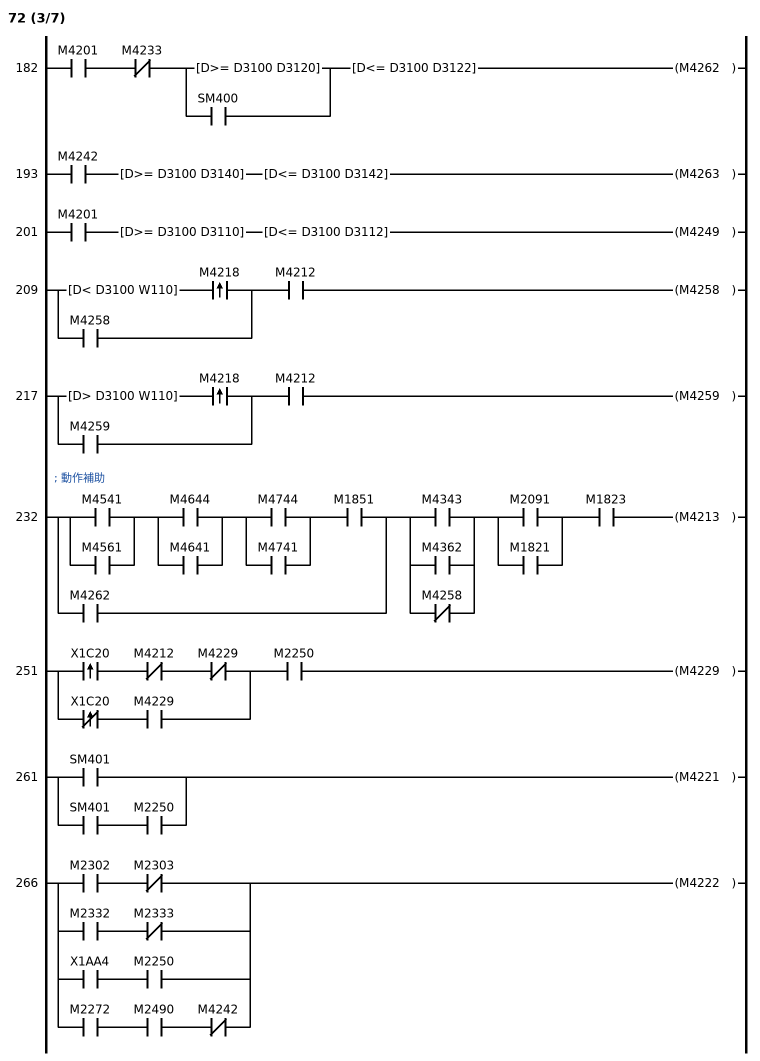
182   LD      M4201
      ANI     M4233
      LDD>=   D3100 D3120
      OR      SM400
      ANB
      ANDD<=  D3100 D3122
      OUT     M4262
193   LD      M4242
      ANDD>=  D3100 D3140
      ANDD<=  D3100 D3142
      OUT     M4263
201   LD      M4201
      ANDD>=  D3100 D3110
      ANDD<=  D3100 D3112
      OUT     M4249
209   LDD<    D3100 W110
      ANDP    M4218
      OR      M4258
      AND     M4212
      OUT     M4258
217   LDD>    D3100 W110
      ANDP    M4218
      OR      M4259
      AND     M4212
      OUT     M4259
; 動作補助
232   LD      M4541
      OR      M4561
      LD      M4644
      OR      M4641
      ANB
      LD      M4744
      OR      M4741
      ANB
      AND     M1851
      OR      M4262
      LD      M4343
      OR      M4362
      ORI     M4258
      ANB
      LD      M2091
      OR      M1821
      ANB
      AND     M1823
      OUT     M4213
251   LDP     X1C20
      ANI     M4212
      ANI     M4229
      LDPI    X1C20
      AND     M4229
      ORB
      AND     M2250
      OUT     M4229
261   LD      SM401
      LD      SM401
      AND     M2250
      ORB
      OUT     M4221
266   LD      M2302
      ANI     M2303
      LD      M2332
      ANI     M2333
      ORB
      LD      X1AA4
      AND     M2250
      ORB
      LD      M2272
      AND     M2490
      ANI     M4242
      ORB
      OUT     M4222
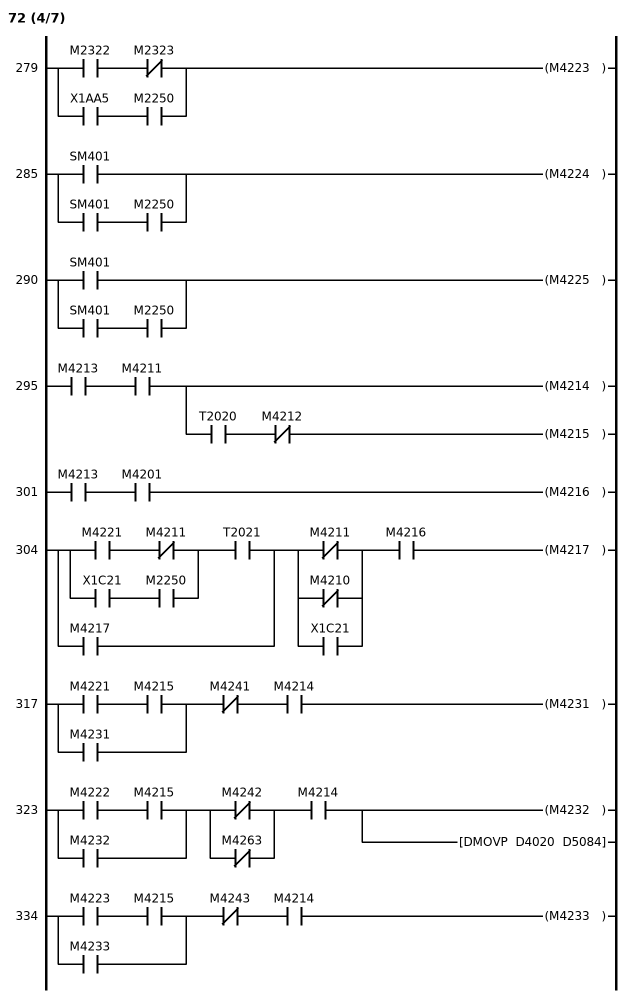
279   LD      M2322
      ANI     M2323
      LD      X1AA5
      AND     M2250
      ORB
      OUT     M4223
285   LD      SM401
      LD      SM401
      AND     M2250
      ORB
      OUT     M4224
290   LD      SM401
      LD      SM401
      AND     M2250
      ORB
      OUT     M4225
295   LD      M4213
      AND     M4211
      OUT     M4214
      AND     T2020
      ANI     M4212
      OUT     M4215
301   LD      M4213
      AND     M4201
      OUT     M4216
304   LD      M4221
      ANI     M4211
      LD      X1C21
      AND     M2250
      ORB
      AND     T2021
      OR      M4217
      LDI     M4211
      ORI     M4210
      OR      X1C21
      ANB
      AND     M4216
      OUT     M4217
317   LD      M4221
      AND     M4215
      OR      M4231
      ANI     M4241
      AND     M4214
      OUT     M4231
323   LD      M4222
      AND     M4215
      OR      M4232
      LDI     M4242
      ORI     M4263
      ANB
      AND     M4214
      OUT     M4232
      DMOVP   D4020 D5084
334   LD      M4223
      AND     M4215
      OR      M4233
      ANI     M4243
      AND     M4214
      OUT     M4233
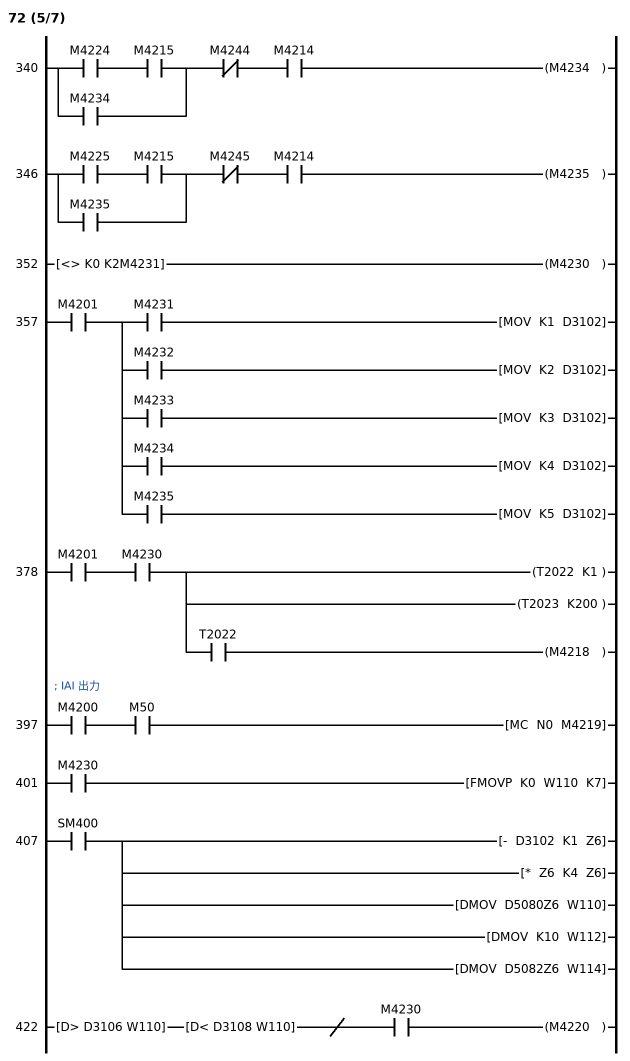
340   LD      M4224
      AND     M4215
      OR      M4234
      ANI     M4244
      AND     M4214
      OUT     M4234
346   LD      M4225
      AND     M4215
      OR      M4235
      ANI     M4245
      AND     M4214
      OUT     M4235
352   LD<>    K0 K2M4231
      OUT     M4230
357   LD      M4201
      MPS
      AND     M4231
      MOV     K1 D3102
      MRD
      AND     M4232
      MOV     K2 D3102
      MRD
      AND     M4233
      MOV     K3 D3102
      MRD
      AND     M4234
      MOV     K4 D3102
      MPP
      AND     M4235
      MOV     K5 D3102
378   LD      M4201
      AND     M4230
      OUT     T2022 K1
      OUT     T2023 K200
      AND     T2022
      OUT     M4218
; IAI 出力
397   LD      M4200
      AND     M50
      MC      N0 M4219
401   LD      M4230
      FMOVP   K0 W110 K7
407   LD      SM400
      -       D3102 K1 Z6
      *       Z6 K4 Z6
      DMOV    D5080Z6 W110
      DMOV    K10 W112
      DMOV    D5082Z6 W114
422   LDD>    D3106 W110
      ANDD<   D3108 W110
      INV
      AND     M4230
      OUT     M4220
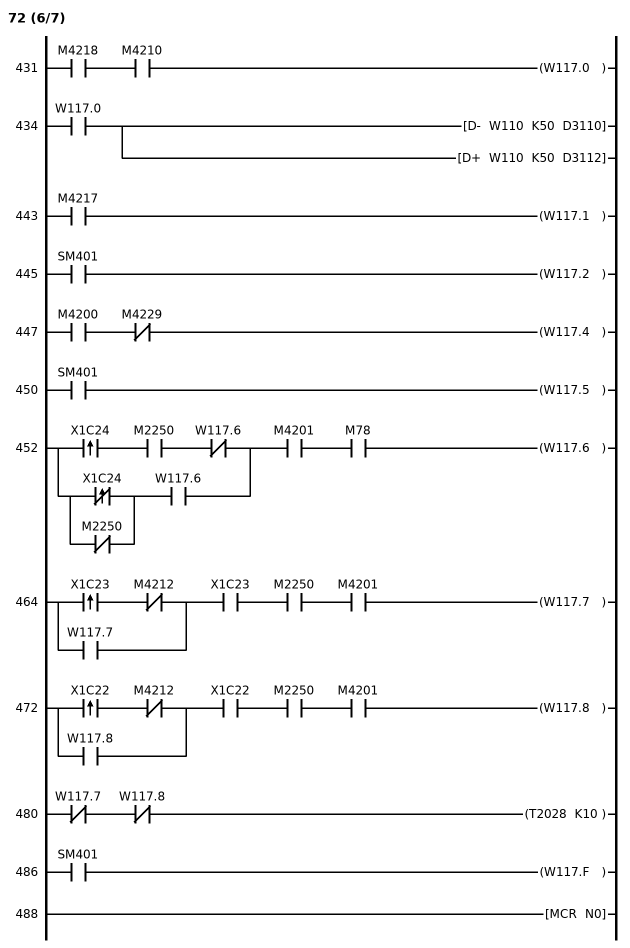
431   LD      M4218
      AND     M4210
      OUT     W117.0
434   LD      W117.0
      D-      W110 K50 D3110
      D+      W110 K50 D3112
443   LD      M4217
      OUT     W117.1
445   LD      SM401
      OUT     W117.2
447   LD      M4200
      ANI     M4229
      OUT     W117.4
450   LD      SM401
      OUT     W117.5
452   LDP     X1C24
      AND     M2250
      ANI     W117.6
      LDPI    X1C24
      ORI     M2250
      AND     W117.6
      ORB
      AND     M4201
      AND     M78
      OUT     W117.6
464   LDP     X1C23
      ANI     M4212
      OR      W117.7
      AND     X1C23
      AND     M2250
      AND     M4201
      OUT     W117.7
472   LDP     X1C22
      ANI     M4212
      OR      W117.8
      AND     X1C22
      AND     M2250
      AND     M4201
      OUT     W117.8
480   LDI     W117.7
      ANI     W117.8
      OUT     T2028 K10
486   LD      SM401
      OUT     W117.F
488   MCR     N0
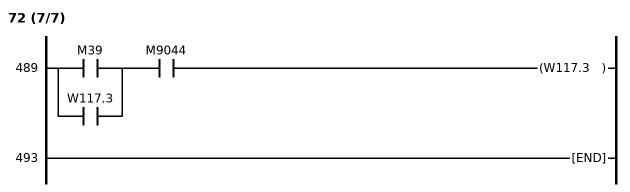
489   LD      M39
      OR      W117.3
      AND     M9044
      OUT     W117.3
493   END
END_PROGRAM

PROGRAM 73
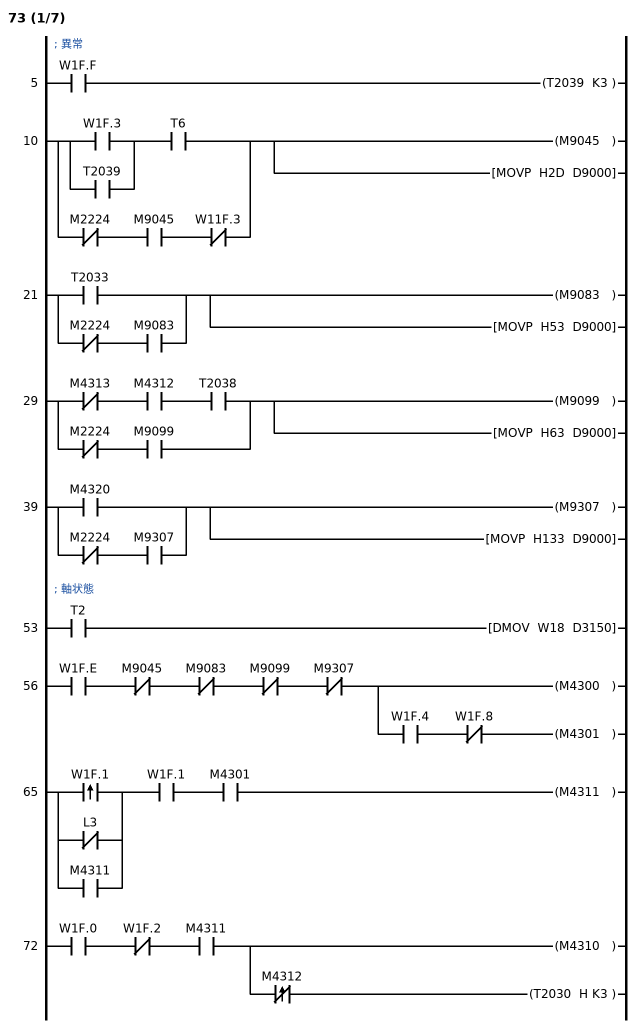
; 異常
5     LD      W1F.F
      OUT     T2039 K3
10    LD      W1F.3
      OR      T2039
      AND     T6
      LDI     M2224
      AND     M9045
      ANI     W11F.3
      ORB
      OUT     M9045
      MOVP    H2D D9000
21    LD      T2033
      LDI     M2224
      AND     M9083
      ORB
      OUT     M9083
      MOVP    H53 D9000
29    LDI     M4313
      AND     M4312
      AND     T2038
      LDI     M2224
      AND     M9099
      ORB
      OUT     M9099
      MOVP    H63 D9000
39    LD      M4320
      LDI     M2224
      AND     M9307
      ORB
      OUT     M9307
      MOVP    H133 D9000
; 軸状態
53    LD      T2
      DMOV    W18 D3150
56    LD      W1F.E
      ANI     M9045
      ANI     M9083
      ANI     M9099
      ANI     M9307
      OUT     M4300
      AND     W1F.4
      ANI     W1F.8
      OUT     M4301
65    LDP     W1F.1
      ORI     L3
      OR      M4311
      AND     W1F.1
      AND     M4301
      OUT     M4311
72    LD      W1F.0
      ANI     W1F.2
      AND     M4311
      OUT     M4310
      ANDPI   M4312
      OUTH    T2030 K3
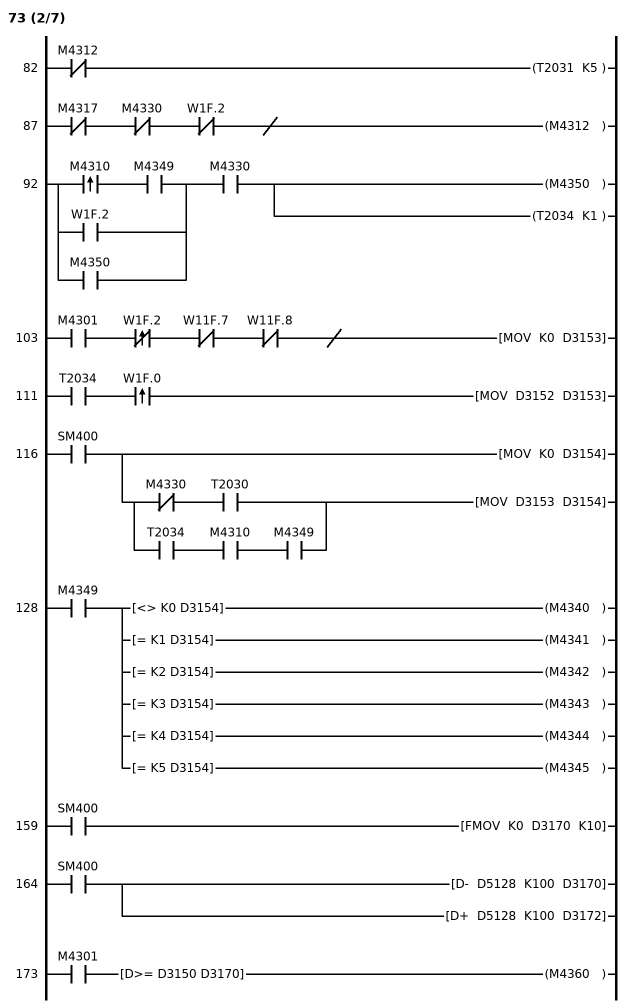
82    LDI     M4312
      OUT     T2031 K5
87    LDI     M4317
      ANI     M4330
      ANI     W1F.2
      INV
      OUT     M4312
92    LDP     M4310
      AND     M4349
      OR      W1F.2
      OR      M4350
      AND     M4330
      OUT     M4350
      OUT     T2034 K1
103   LD      M4301
      ANDPI   W1F.2
      ANI     W11F.7
      ANI     W11F.8
      INV
      MOV     K0 D3153
111   LD      T2034
      ANDP    W1F.0
      MOV     D3152 D3153
116   LD      SM400
      MOV     K0 D3154
      LDI     M4330
      AND     T2030
      LD      T2034
      AND     M4310
      AND     M4349
      ORB
      ANB
      MOV     D3153 D3154
128   LD      M4349
      MPS
      AND<>   K0 D3154
      OUT     M4340
      MRD
      AND=    K1 D3154
      OUT     M4341
      MRD
      AND=    K2 D3154
      OUT     M4342
      MRD
      AND=    K3 D3154
      OUT     M4343
      MRD
      AND=    K4 D3154
      OUT     M4344
      MPP
      AND=    K5 D3154
      OUT     M4345
159   LD      SM400
      FMOV    K0 D3170 K10
164   LD      SM400
      D-      D5128 K100 D3170
      D+      D5128 K100 D3172
173   LD      M4301
      ANDD>=  D3150 D3170
      OUT     M4360
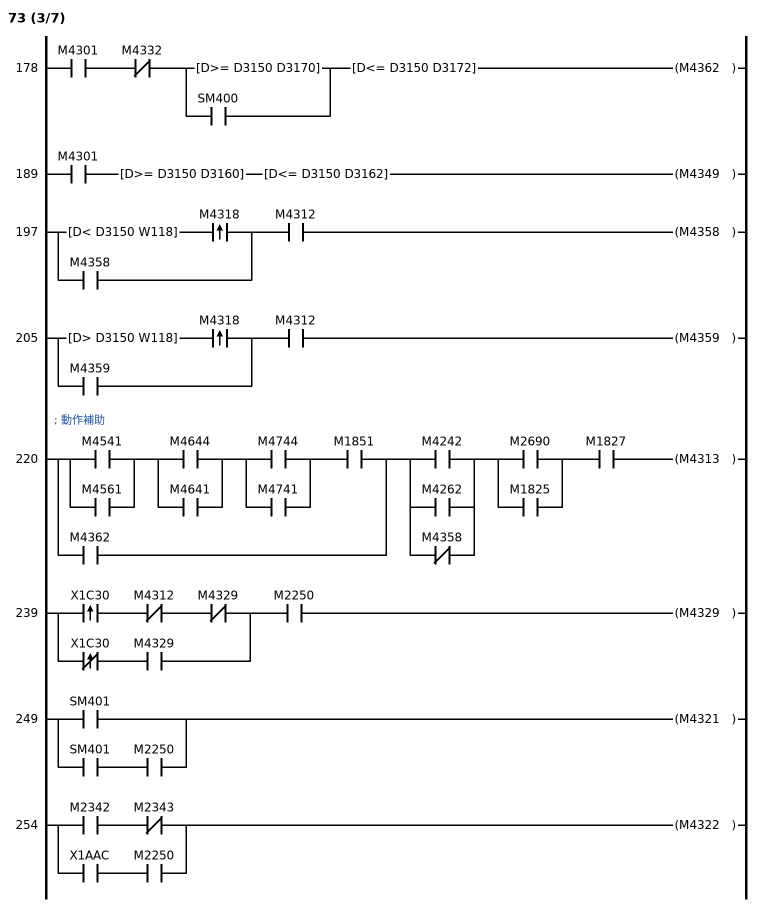
178   LD      M4301
      ANI     M4332
      LDD>=   D3150 D3170
      OR      SM400
      ANB
      ANDD<=  D3150 D3172
      OUT     M4362
189   LD      M4301
      ANDD>=  D3150 D3160
      ANDD<=  D3150 D3162
      OUT     M4349
197   LDD<    D3150 W118
      ANDP    M4318
      OR      M4358
      AND     M4312
      OUT     M4358
205   LDD>    D3150 W118
      ANDP    M4318
      OR      M4359
      AND     M4312
      OUT     M4359
; 動作補助
220   LD      M4541
      OR      M4561
      LD      M4644
      OR      M4641
      ANB
      LD      M4744
      OR      M4741
      ANB
      AND     M1851
      OR      M4362
      LD      M4242
      OR      M4262
      ORI     M4358
      ANB
      LD      M2690
      OR      M1825
      ANB
      AND     M1827
      OUT     M4313
239   LDP     X1C30
      ANI     M4312
      ANI     M4329
      LDPI    X1C30
      AND     M4329
      ORB
      AND     M2250
      OUT     M4329
249   LD      SM401
      LD      SM401
      AND     M2250
      ORB
      OUT     M4321
254   LD      M2342
      ANI     M2343
      LD      X1AAC
      AND     M2250
      ORB
      OUT     M4322
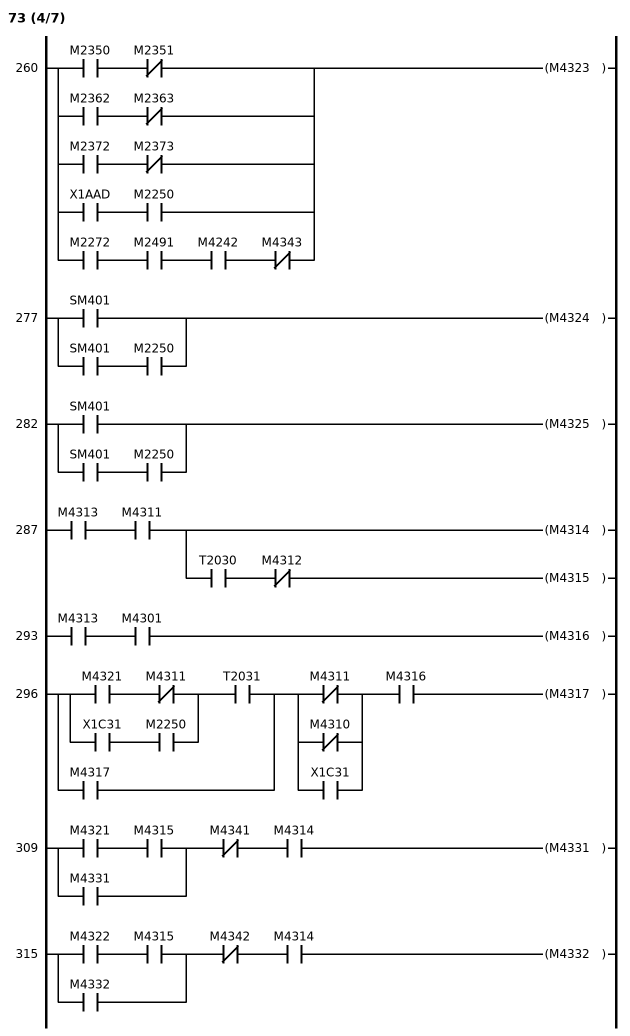
260   LD      M2350
      ANI     M2351
      LD      M2362
      ANI     M2363
      ORB
      LD      M2372
      ANI     M2373
      ORB
      LD      X1AAD
      AND     M2250
      ORB
      LD      M2272
      AND     M2491
      AND     M4242
      ANI     M4343
      ORB
      OUT     M4323
277   LD      SM401
      LD      SM401
      AND     M2250
      ORB
      OUT     M4324
282   LD      SM401
      LD      SM401
      AND     M2250
      ORB
      OUT     M4325
287   LD      M4313
      AND     M4311
      OUT     M4314
      AND     T2030
      ANI     M4312
      OUT     M4315
293   LD      M4313
      AND     M4301
      OUT     M4316
296   LD      M4321
      ANI     M4311
      LD      X1C31
      AND     M2250
      ORB
      AND     T2031
      OR      M4317
      LDI     M4311
      ORI     M4310
      OR      X1C31
      ANB
      AND     M4316
      OUT     M4317
309   LD      M4321
      AND     M4315
      OR      M4331
      ANI     M4341
      AND     M4314
      OUT     M4331
315   LD      M4322
      AND     M4315
      OR      M4332
      ANI     M4342
      AND     M4314
      OUT     M4332
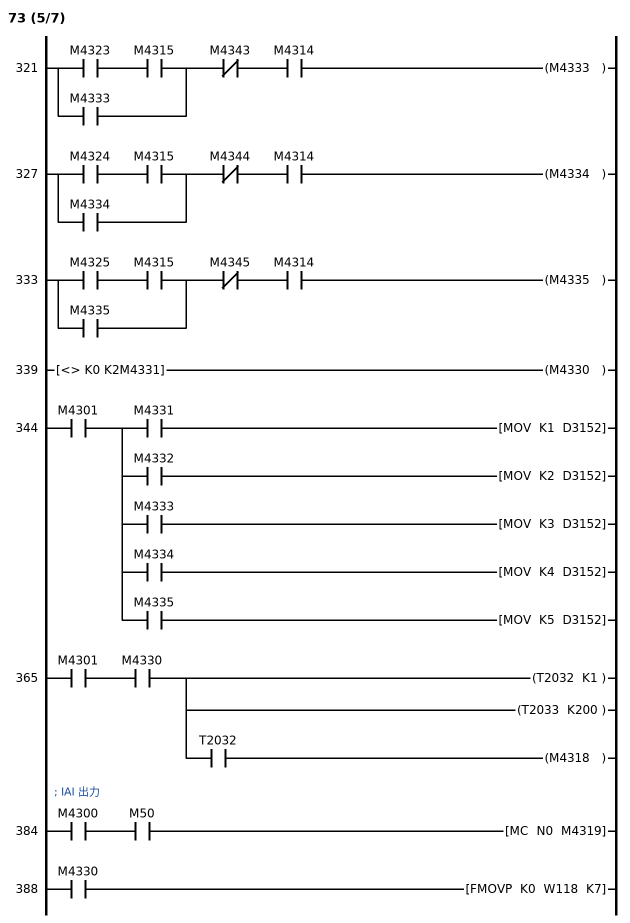
321   LD      M4323
      AND     M4315
      OR      M4333
      ANI     M4343
      AND     M4314
      OUT     M4333
327   LD      M4324
      AND     M4315
      OR      M4334
      ANI     M4344
      AND     M4314
      OUT     M4334
333   LD      M4325
      AND     M4315
      OR      M4335
      ANI     M4345
      AND     M4314
      OUT     M4335
339   LD<>    K0 K2M4331
      OUT     M4330
344   LD      M4301
      MPS
      AND     M4331
      MOV     K1 D3152
      MRD
      AND     M4332
      MOV     K2 D3152
      MRD
      AND     M4333
      MOV     K3 D3152
      MRD
      AND     M4334
      MOV     K4 D3152
      MPP
      AND     M4335
      MOV     K5 D3152
365   LD      M4301
      AND     M4330
      OUT     T2032 K1
      OUT     T2033 K200
      AND     T2032
      OUT     M4318
; IAI 出力
384   LD      M4300
      AND     M50
      MC      N0 M4319
388   LD      M4330
      FMOVP   K0 W118 K7
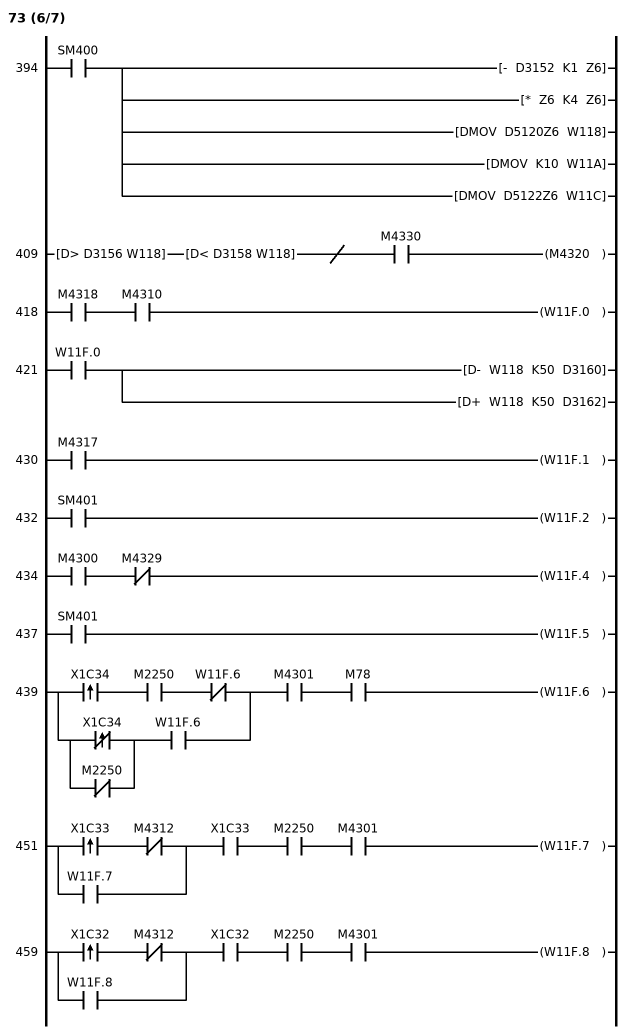
394   LD      SM400
      -       D3152 K1 Z6
      *       Z6 K4 Z6
      DMOV    D5120Z6 W118
      DMOV    K10 W11A
      DMOV    D5122Z6 W11C
409   LDD>    D3156 W118
      ANDD<   D3158 W118
      INV
      AND     M4330
      OUT     M4320
418   LD      M4318
      AND     M4310
      OUT     W11F.0
421   LD      W11F.0
      D-      W118 K50 D3160
      D+      W118 K50 D3162
430   LD      M4317
      OUT     W11F.1
432   LD      SM401
      OUT     W11F.2
434   LD      M4300
      ANI     M4329
      OUT     W11F.4
437   LD      SM401
      OUT     W11F.5
439   LDP     X1C34
      AND     M2250
      ANI     W11F.6
      LDPI    X1C34
      ORI     M2250
      AND     W11F.6
      ORB
      AND     M4301
      AND     M78
      OUT     W11F.6
451   LDP     X1C33
      ANI     M4312
      OR      W11F.7
      AND     X1C33
      AND     M2250
      AND     M4301
      OUT     W11F.7
459   LDP     X1C32
      ANI     M4312
      OR      W11F.8
      AND     X1C32
      AND     M2250
      AND     M4301
      OUT     W11F.8
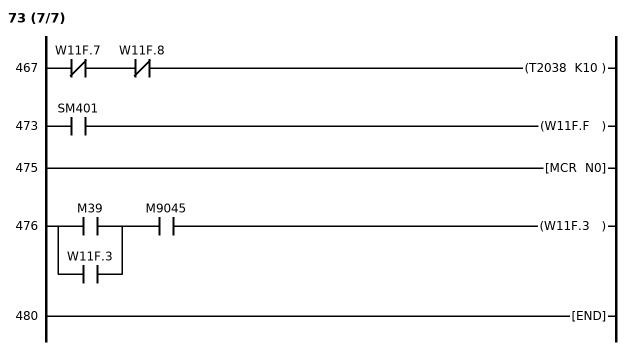
467   LDI     W11F.7
      ANI     W11F.8
      OUT     T2038 K10
473   LD      SM401
      OUT     W11F.F
475   MCR     N0
476   LD      M39
      OR      W11F.3
      AND     M9045
      OUT     W11F.3
480   END
END_PROGRAM

PROGRAM 74
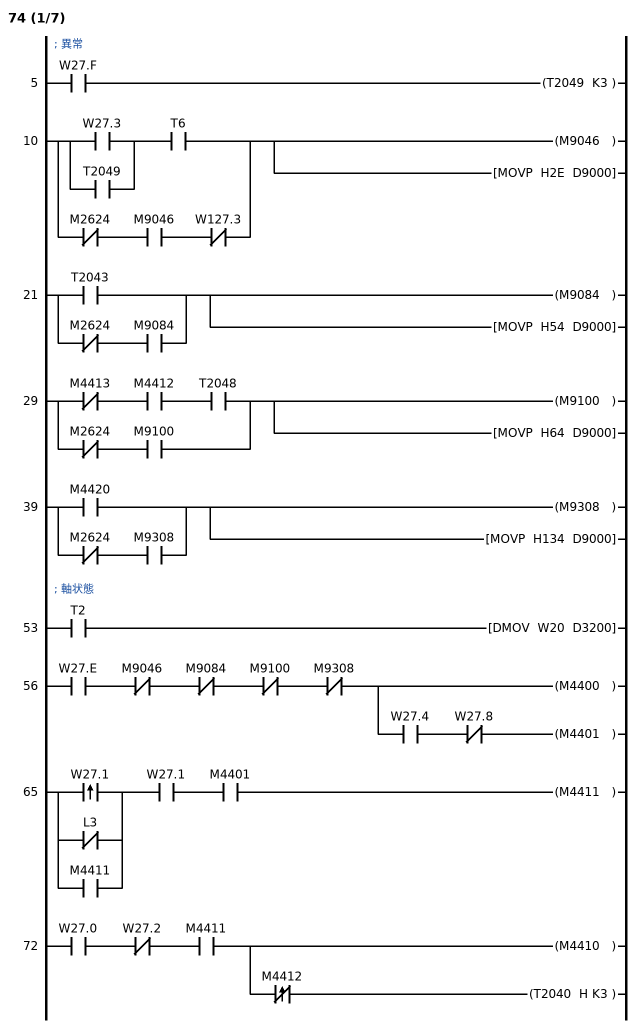
; 異常
5     LD      W27.F
      OUT     T2049 K3
10    LD      W27.3
      OR      T2049
      AND     T6
      LDI     M2624
      AND     M9046
      ANI     W127.3
      ORB
      OUT     M9046
      MOVP    H2E D9000
21    LD      T2043
      LDI     M2624
      AND     M9084
      ORB
      OUT     M9084
      MOVP    H54 D9000
29    LDI     M4413
      AND     M4412
      AND     T2048
      LDI     M2624
      AND     M9100
      ORB
      OUT     M9100
      MOVP    H64 D9000
39    LD      M4420
      LDI     M2624
      AND     M9308
      ORB
      OUT     M9308
      MOVP    H134 D9000
; 軸状態
53    LD      T2
      DMOV    W20 D3200
56    LD      W27.E
      ANI     M9046
      ANI     M9084
      ANI     M9100
      ANI     M9308
      OUT     M4400
      AND     W27.4
      ANI     W27.8
      OUT     M4401
65    LDP     W27.1
      ORI     L3
      OR      M4411
      AND     W27.1
      AND     M4401
      OUT     M4411
72    LD      W27.0
      ANI     W27.2
      AND     M4411
      OUT     M4410
      ANDPI   M4412
      OUTH    T2040 K3
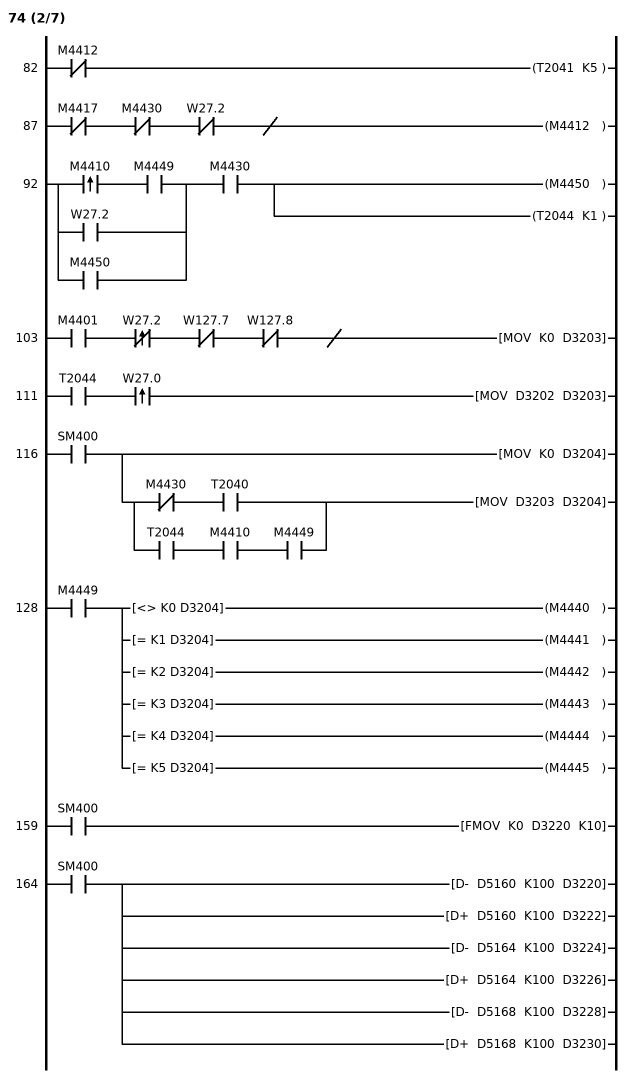
82    LDI     M4412
      OUT     T2041 K5
87    LDI     M4417
      ANI     M4430
      ANI     W27.2
      INV
      OUT     M4412
92    LDP     M4410
      AND     M4449
      OR      W27.2
      OR      M4450
      AND     M4430
      OUT     M4450
      OUT     T2044 K1
103   LD      M4401
      ANDPI   W27.2
      ANI     W127.7
      ANI     W127.8
      INV
      MOV     K0 D3203
111   LD      T2044
      ANDP    W27.0
      MOV     D3202 D3203
116   LD      SM400
      MOV     K0 D3204
      LDI     M4430
      AND     T2040
      LD      T2044
      AND     M4410
      AND     M4449
      ORB
      ANB
      MOV     D3203 D3204
128   LD      M4449
      MPS
      AND<>   K0 D3204
      OUT     M4440
      MRD
      AND=    K1 D3204
      OUT     M4441
      MRD
      AND=    K2 D3204
      OUT     M4442
      MRD
      AND=    K3 D3204
      OUT     M4443
      MRD
      AND=    K4 D3204
      OUT     M4444
      MPP
      AND=    K5 D3204
      OUT     M4445
159   LD      SM400
      FMOV    K0 D3220 K10
164   LD      SM400
      D-      D5160 K100 D3220
      D+      D5160 K100 D3222
      D-      D5164 K100 D3224
      D+      D5164 K100 D3226
      D-      D5168 K100 D3228
      D+      D5168 K100 D3230
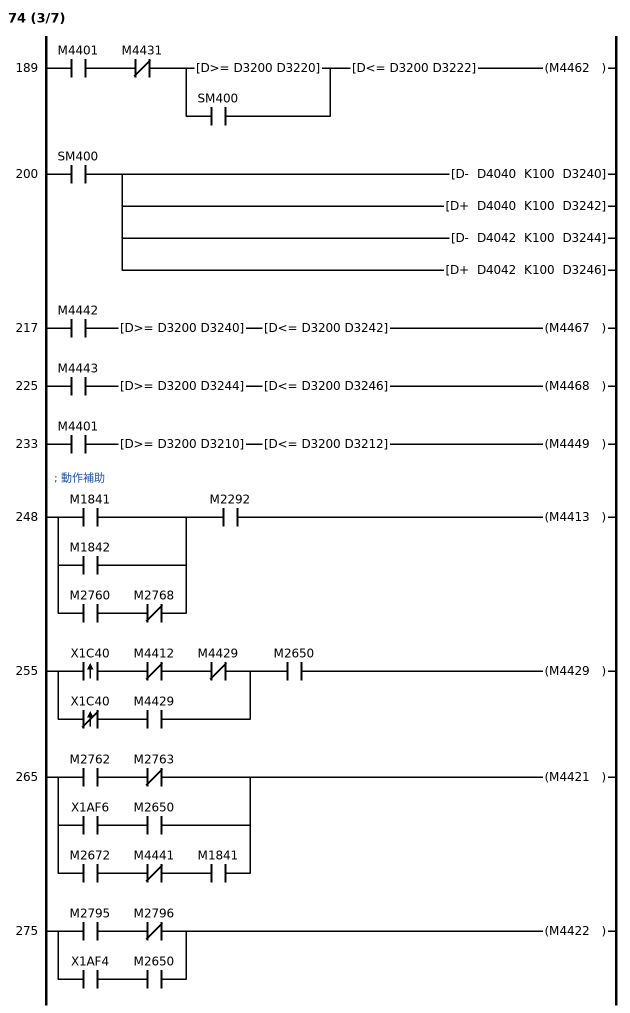
189   LD      M4401
      ANI     M4431
      LDD>=   D3200 D3220
      OR      SM400
      ANB
      ANDD<=  D3200 D3222
      OUT     M4462
200   LD      SM400
      D-      D4040 K100 D3240
      D+      D4040 K100 D3242
      D-      D4042 K100 D3244
      D+      D4042 K100 D3246
217   LD      M4442
      ANDD>=  D3200 D3240
      ANDD<=  D3200 D3242
      OUT     M4467
225   LD      M4443
      ANDD>=  D3200 D3244
      ANDD<=  D3200 D3246
      OUT     M4468
233   LD      M4401
      ANDD>=  D3200 D3210
      ANDD<=  D3200 D3212
      OUT     M4449
; 動作補助
248   LD      M1841
      OR      M1842
      LD      M2760
      ANI     M2768
      ORB
      AND     M2292
      OUT     M4413
255   LDP     X1C40
      ANI     M4412
      ANI     M4429
      LDPI    X1C40
      AND     M4429
      ORB
      AND     M2650
      OUT     M4429
265   LD      M2762
      ANI     M2763
      LD      X1AF6
      AND     M2650
      ORB
      LD      M2672
      ANI     M4441
      AND     M1841
      ORB
      OUT     M4421
275   LD      M2795
      ANI     M2796
      LD      X1AF4
      AND     M2650
      ORB
      OUT     M4422
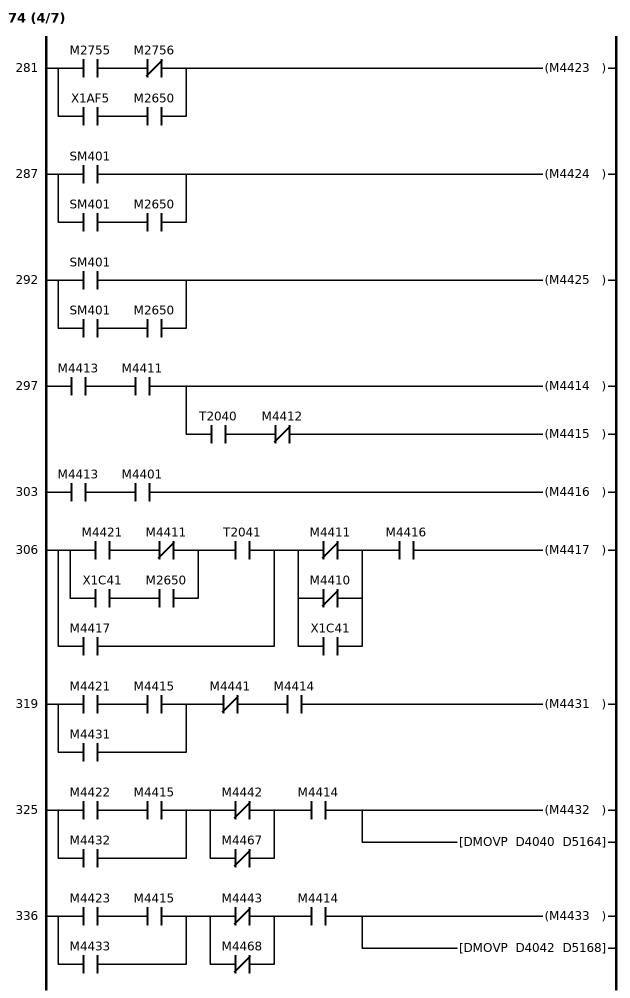
281   LD      M2755
      ANI     M2756
      LD      X1AF5
      AND     M2650
      ORB
      OUT     M4423
287   LD      SM401
      LD      SM401
      AND     M2650
      ORB
      OUT     M4424
292   LD      SM401
      LD      SM401
      AND     M2650
      ORB
      OUT     M4425
297   LD      M4413
      AND     M4411
      OUT     M4414
      AND     T2040
      ANI     M4412
      OUT     M4415
303   LD      M4413
      AND     M4401
      OUT     M4416
306   LD      M4421
      ANI     M4411
      LD      X1C41
      AND     M2650
      ORB
      AND     T2041
      OR      M4417
      LDI     M4411
      ORI     M4410
      OR      X1C41
      ANB
      AND     M4416
      OUT     M4417
319   LD      M4421
      AND     M4415
      OR      M4431
      ANI     M4441
      AND     M4414
      OUT     M4431
325   LD      M4422
      AND     M4415
      OR      M4432
      LDI     M4442
      ORI     M4467
      ANB
      AND     M4414
      OUT     M4432
      DMOVP   D4040 D5164
336   LD      M4423
      AND     M4415
      OR      M4433
      LDI     M4443
      ORI     M4468
      ANB
      AND     M4414
      OUT     M4433
      DMOVP   D4042 D5168
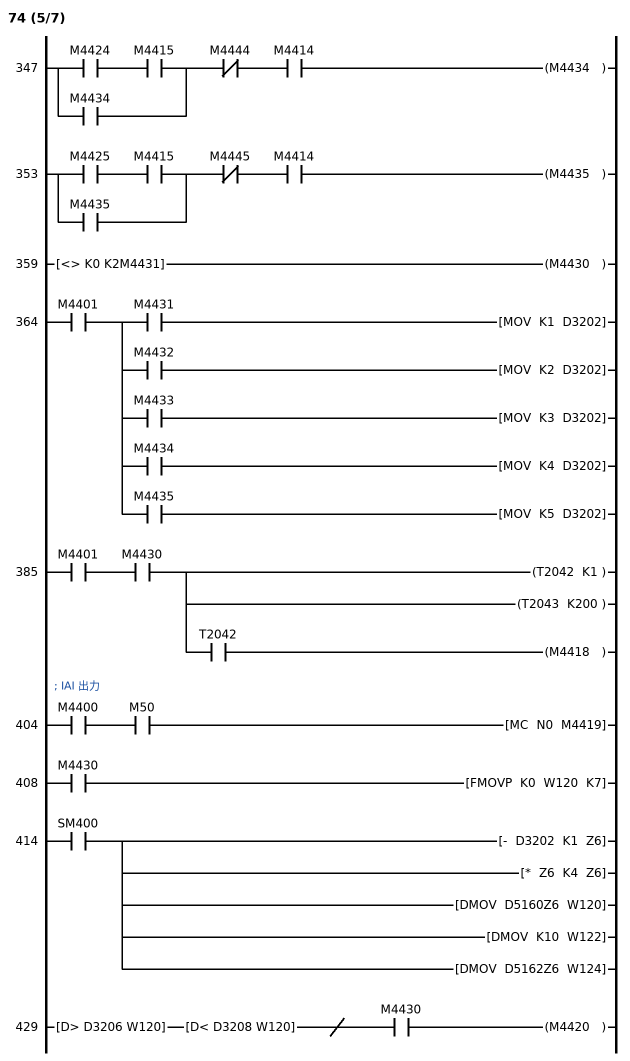
347   LD      M4424
      AND     M4415
      OR      M4434
      ANI     M4444
      AND     M4414
      OUT     M4434
353   LD      M4425
      AND     M4415
      OR      M4435
      ANI     M4445
      AND     M4414
      OUT     M4435
359   LD<>    K0 K2M4431
      OUT     M4430
364   LD      M4401
      MPS
      AND     M4431
      MOV     K1 D3202
      MRD
      AND     M4432
      MOV     K2 D3202
      MRD
      AND     M4433
      MOV     K3 D3202
      MRD
      AND     M4434
      MOV     K4 D3202
      MPP
      AND     M4435
      MOV     K5 D3202
385   LD      M4401
      AND     M4430
      OUT     T2042 K1
      OUT     T2043 K200
      AND     T2042
      OUT     M4418
; IAI 出力
404   LD      M4400
      AND     M50
      MC      N0 M4419
408   LD      M4430
      FMOVP   K0 W120 K7
414   LD      SM400
      -       D3202 K1 Z6
      *       Z6 K4 Z6
      DMOV    D5160Z6 W120
      DMOV    K10 W122
      DMOV    D5162Z6 W124
429   LDD>    D3206 W120
      ANDD<   D3208 W120
      INV
      AND     M4430
      OUT     M4420
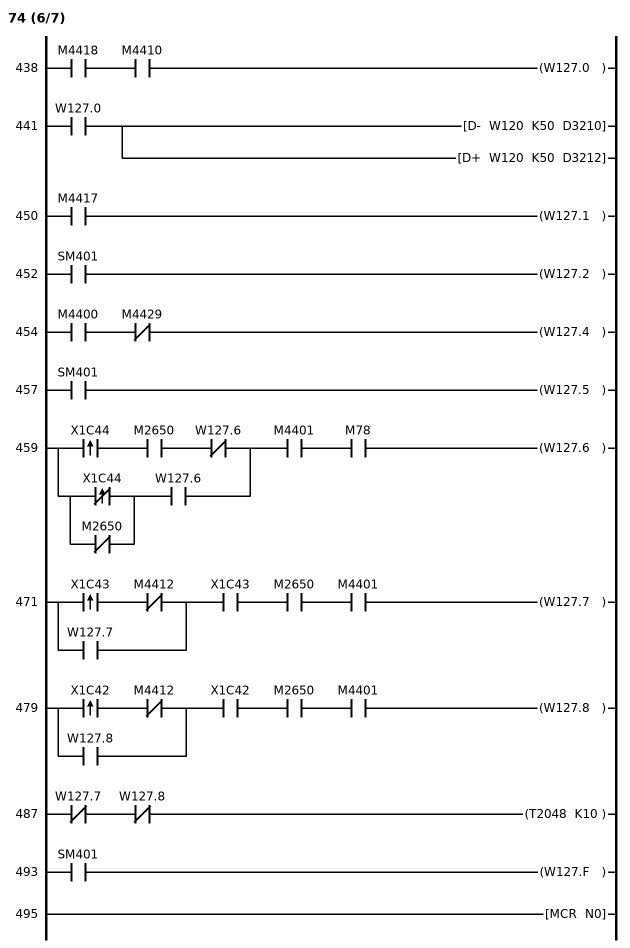
438   LD      M4418
      AND     M4410
      OUT     W127.0
441   LD      W127.0
      D-      W120 K50 D3210
      D+      W120 K50 D3212
450   LD      M4417
      OUT     W127.1
452   LD      SM401
      OUT     W127.2
454   LD      M4400
      ANI     M4429
      OUT     W127.4
457   LD      SM401
      OUT     W127.5
459   LDP     X1C44
      AND     M2650
      ANI     W127.6
      LDPI    X1C44
      ORI     M2650
      AND     W127.6
      ORB
      AND     M4401
      AND     M78
      OUT     W127.6
471   LDP     X1C43
      ANI     M4412
      OR      W127.7
      AND     X1C43
      AND     M2650
      AND     M4401
      OUT     W127.7
479   LDP     X1C42
      ANI     M4412
      OR      W127.8
      AND     X1C42
      AND     M2650
      AND     M4401
      OUT     W127.8
487   LDI     W127.7
      ANI     W127.8
      OUT     T2048 K10
493   LD      SM401
      OUT     W127.F
495   MCR     N0
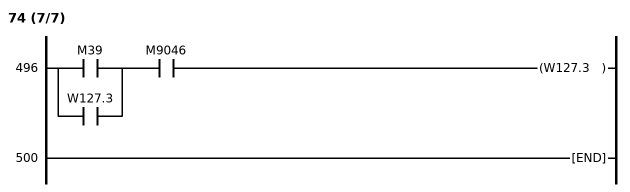
496   LD      M39
      OR      W127.3
      AND     M9046
      OUT     W127.3
500   END
END_PROGRAM

PROGRAM 75
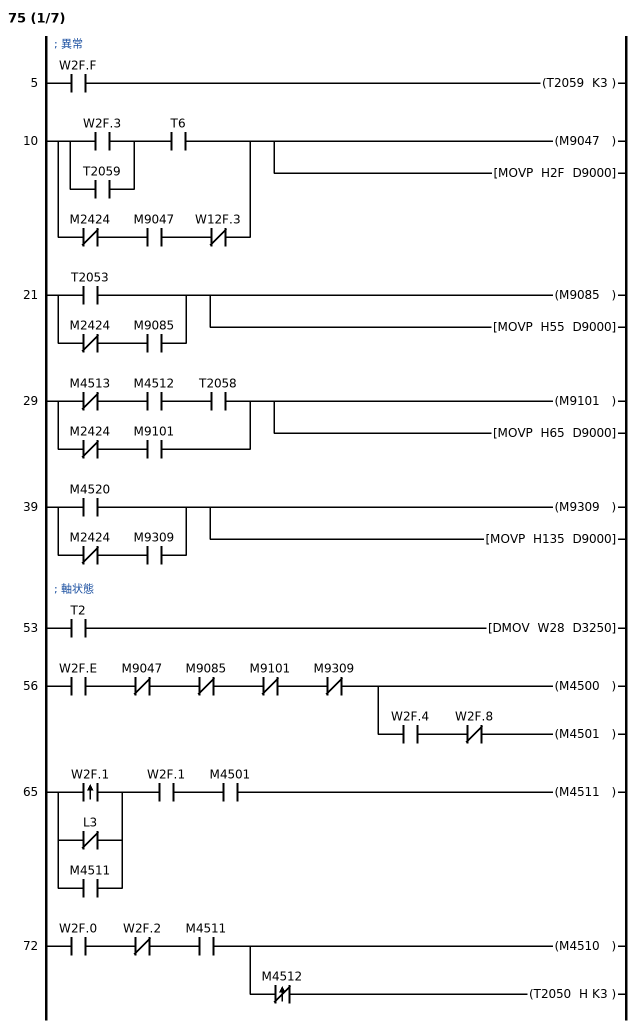
; 異常
5     LD      W2F.F
      OUT     T2059 K3
10    LD      W2F.3
      OR      T2059
      AND     T6
      LDI     M2424
      AND     M9047
      ANI     W12F.3
      ORB
      OUT     M9047
      MOVP    H2F D9000
21    LD      T2053
      LDI     M2424
      AND     M9085
      ORB
      OUT     M9085
      MOVP    H55 D9000
29    LDI     M4513
      AND     M4512
      AND     T2058
      LDI     M2424
      AND     M9101
      ORB
      OUT     M9101
      MOVP    H65 D9000
39    LD      M4520
      LDI     M2424
      AND     M9309
      ORB
      OUT     M9309
      MOVP    H135 D9000
; 軸状態
53    LD      T2
      DMOV    W28 D3250
56    LD      W2F.E
      ANI     M9047
      ANI     M9085
      ANI     M9101
      ANI     M9309
      OUT     M4500
      AND     W2F.4
      ANI     W2F.8
      OUT     M4501
65    LDP     W2F.1
      ORI     L3
      OR      M4511
      AND     W2F.1
      AND     M4501
      OUT     M4511
72    LD      W2F.0
      ANI     W2F.2
      AND     M4511
      OUT     M4510
      ANDPI   M4512
      OUTH    T2050 K3
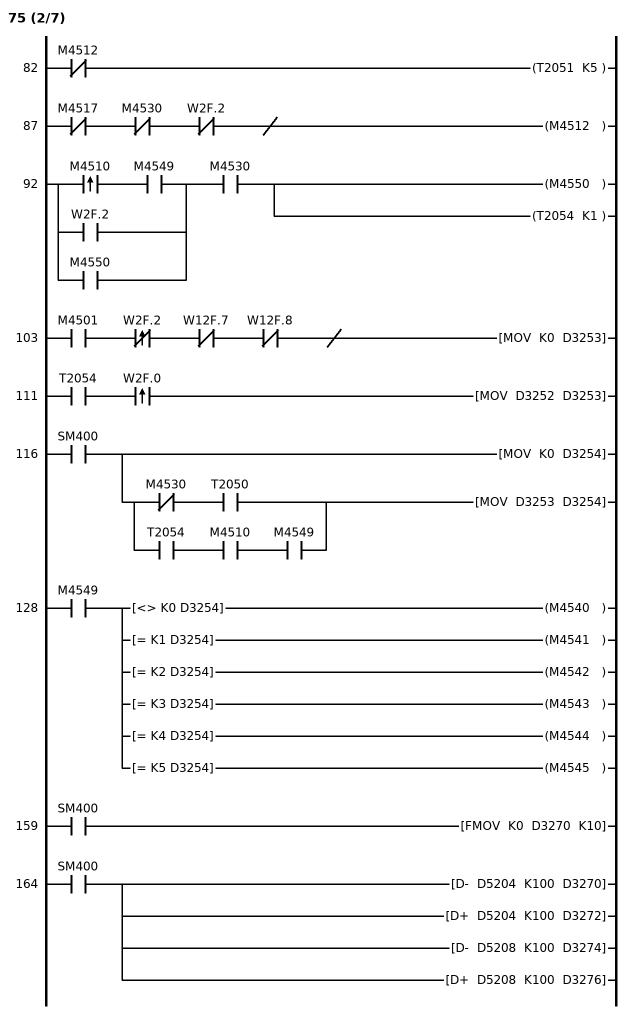
82    LDI     M4512
      OUT     T2051 K5
87    LDI     M4517
      ANI     M4530
      ANI     W2F.2
      INV
      OUT     M4512
92    LDP     M4510
      AND     M4549
      OR      W2F.2
      OR      M4550
      AND     M4530
      OUT     M4550
      OUT     T2054 K1
103   LD      M4501
      ANDPI   W2F.2
      ANI     W12F.7
      ANI     W12F.8
      INV
      MOV     K0 D3253
111   LD      T2054
      ANDP    W2F.0
      MOV     D3252 D3253
116   LD      SM400
      MOV     K0 D3254
      LDI     M4530
      AND     T2050
      LD      T2054
      AND     M4510
      AND     M4549
      ORB
      ANB
      MOV     D3253 D3254
128   LD      M4549
      MPS
      AND<>   K0 D3254
      OUT     M4540
      MRD
      AND=    K1 D3254
      OUT     M4541
      MRD
      AND=    K2 D3254
      OUT     M4542
      MRD
      AND=    K3 D3254
      OUT     M4543
      MRD
      AND=    K4 D3254
      OUT     M4544
      MPP
      AND=    K5 D3254
      OUT     M4545
159   LD      SM400
      FMOV    K0 D3270 K10
164   LD      SM400
      D-      D5204 K100 D3270
      D+      D5204 K100 D3272
      D-      D5208 K100 D3274
      D+      D5208 K100 D3276
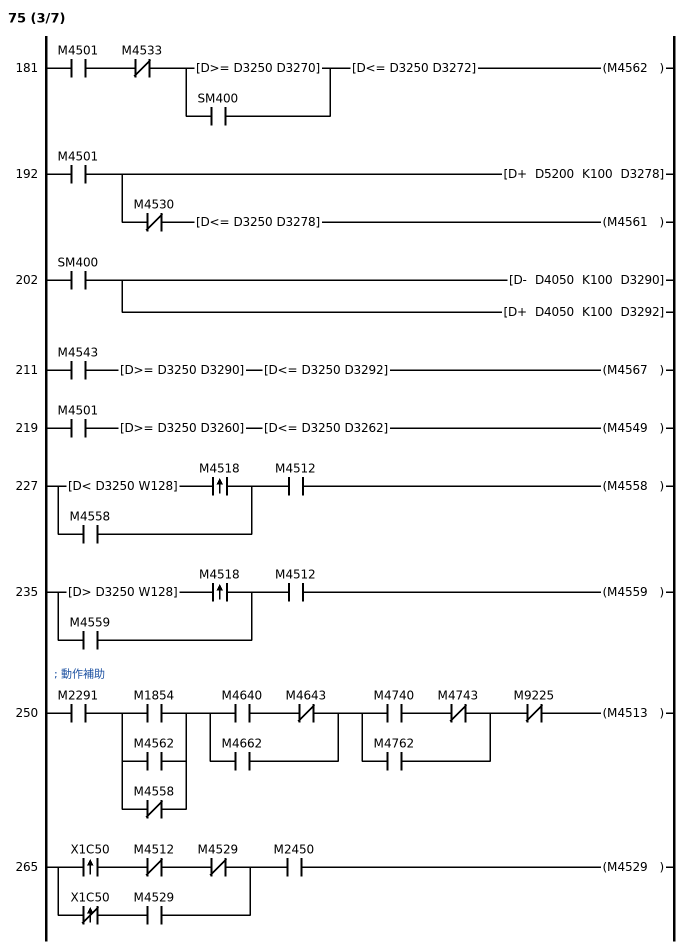
181   LD      M4501
      ANI     M4533
      LDD>=   D3250 D3270
      OR      SM400
      ANB
      ANDD<=  D3250 D3272
      OUT     M4562
192   LD      M4501
      D+      D5200 K100 D3278
      ANI     M4530
      ANDD<=  D3250 D3278
      OUT     M4561
202   LD      SM400
      D-      D4050 K100 D3290
      D+      D4050 K100 D3292
211   LD      M4543
      ANDD>=  D3250 D3290
      ANDD<=  D3250 D3292
      OUT     M4567
219   LD      M4501
      ANDD>=  D3250 D3260
      ANDD<=  D3250 D3262
      OUT     M4549
227   LDD<    D3250 W128
      ANDP    M4518
      OR      M4558
      AND     M4512
      OUT     M4558
235   LDD>    D3250 W128
      ANDP    M4518
      OR      M4559
      AND     M4512
      OUT     M4559
; 動作補助
250   LD      M2291
      LD      M1854
      OR      M4562
      ORI     M4558
      ANB
      LD      M4640
      ANI     M4643
      OR      M4662
      ANB
      LD      M4740
      ANI     M4743
      OR      M4762
      ANB
      ANI     M9225
      OUT     M4513
265   LDP     X1C50
      ANI     M4512
      ANI     M4529
      LDPI    X1C50
      AND     M4529
      ORB
      AND     M2450
      OUT     M4529
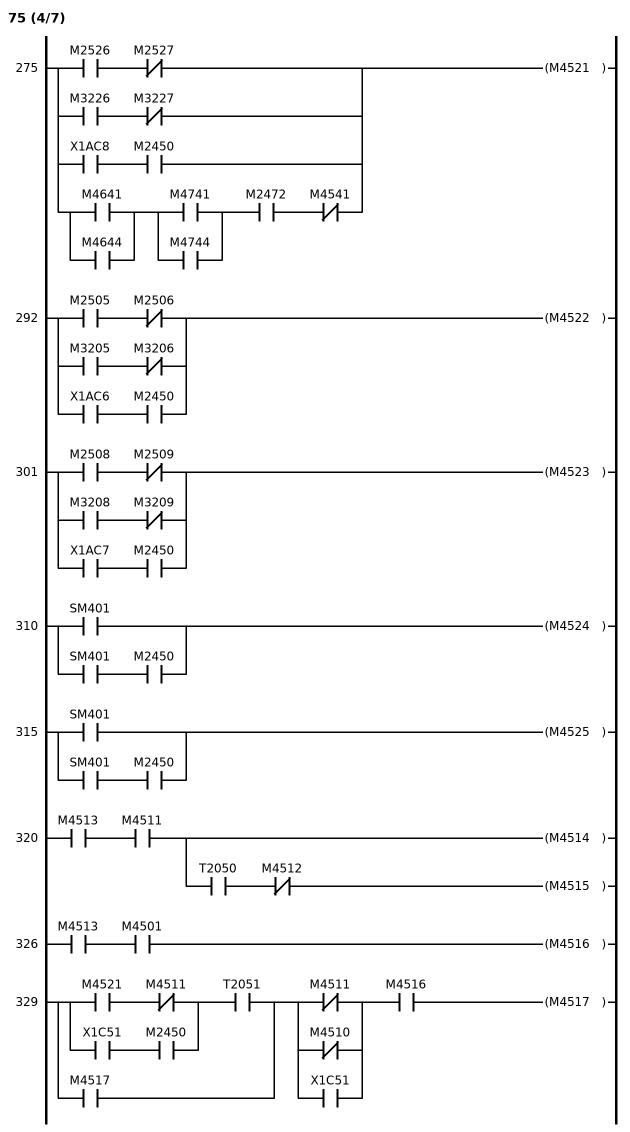
275   LD      M2526
      ANI     M2527
      LD      M3226
      ANI     M3227
      ORB
      LD      X1AC8
      AND     M2450
      ORB
      LD      M4641
      OR      M4644
      LD      M4741
      OR      M4744
      ANB
      AND     M2472
      ANI     M4541
      ORB
      OUT     M4521
292   LD      M2505
      ANI     M2506
      LD      M3205
      ANI     M3206
      ORB
      LD      X1AC6
      AND     M2450
      ORB
      OUT     M4522
301   LD      M2508
      ANI     M2509
      LD      M3208
      ANI     M3209
      ORB
      LD      X1AC7
      AND     M2450
      ORB
      OUT     M4523
310   LD      SM401
      LD      SM401
      AND     M2450
      ORB
      OUT     M4524
315   LD      SM401
      LD      SM401
      AND     M2450
      ORB
      OUT     M4525
320   LD      M4513
      AND     M4511
      OUT     M4514
      AND     T2050
      ANI     M4512
      OUT     M4515
326   LD      M4513
      AND     M4501
      OUT     M4516
329   LD      M4521
      ANI     M4511
      LD      X1C51
      AND     M2450
      ORB
      AND     T2051
      OR      M4517
      LDI     M4511
      ORI     M4510
      OR      X1C51
      ANB
      AND     M4516
      OUT     M4517
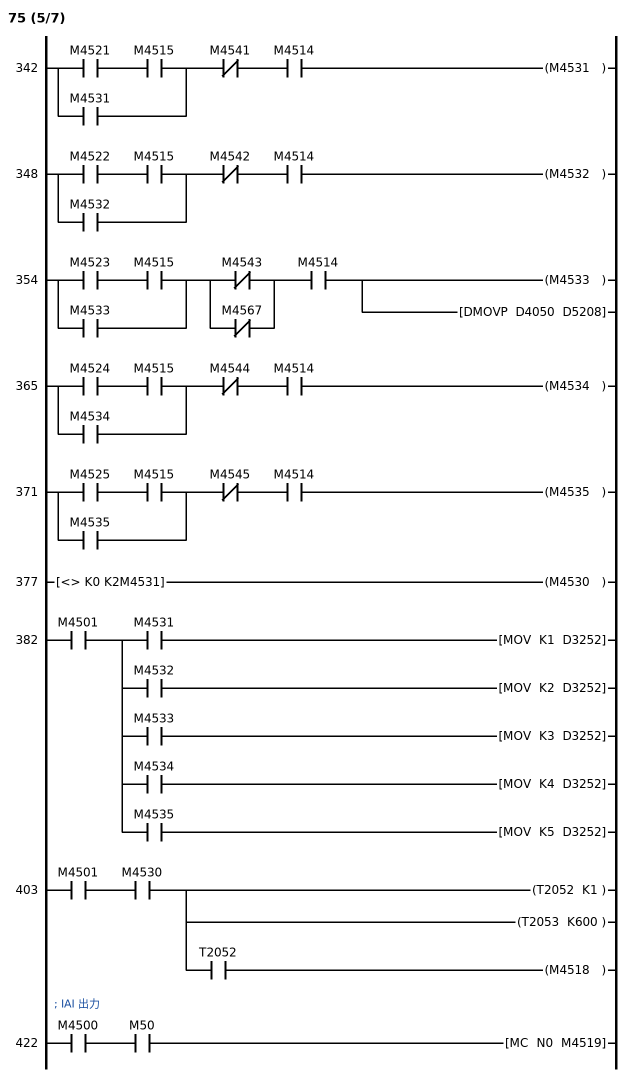
342   LD      M4521
      AND     M4515
      OR      M4531
      ANI     M4541
      AND     M4514
      OUT     M4531
348   LD      M4522
      AND     M4515
      OR      M4532
      ANI     M4542
      AND     M4514
      OUT     M4532
354   LD      M4523
      AND     M4515
      OR      M4533
      LDI     M4543
      ORI     M4567
      ANB
      AND     M4514
      OUT     M4533
      DMOVP   D4050 D5208
365   LD      M4524
      AND     M4515
      OR      M4534
      ANI     M4544
      AND     M4514
      OUT     M4534
371   LD      M4525
      AND     M4515
      OR      M4535
      ANI     M4545
      AND     M4514
      OUT     M4535
377   LD<>    K0 K2M4531
      OUT     M4530
382   LD      M4501
      MPS
      AND     M4531
      MOV     K1 D3252
      MRD
      AND     M4532
      MOV     K2 D3252
      MRD
      AND     M4533
      MOV     K3 D3252
      MRD
      AND     M4534
      MOV     K4 D3252
      MPP
      AND     M4535
      MOV     K5 D3252
403   LD      M4501
      AND     M4530
      OUT     T2052 K1
      OUT     T2053 K600
      AND     T2052
      OUT     M4518
; IAI 出力
422   LD      M4500
      AND     M50
      MC      N0 M4519
